{attribute addProperty BoxType "EPP1342-0001-0017"}
{attribute addProperty Id "A_0025_EPP1518_0002_0016EPP1518_7C3C20DE36846A_0026_EPP1518_0002_0017EPP1518_7C3C20DE36846A_0027_EPP1809_0021_0016EPP1809_8059E62316020A_0028_EPP1809_0022_0016EPP1809_8059E62316020A_0029_EPP1819_0021_0016EPP1819_8059E62316020A_0030_EPP1819_0022_0016EPP1819_8059E62316020A_0031_EPP1816_0003_0016EPP1816_9D1B0E2325632A_0032_EPP1816_0008_0016EPP1816_8EE49DA824030A_0033_EPP1816_0008_0017EPP1816_8EE49DA824030A_0034_EPP1816_0008_0018EPP1816_9D1B0E2325632A_0035_EPP1816_3008_0016EPP1816_5F09590E44856"}
{attribute addProperty CRC "1107668744"}
{attribute addProperty SizeInBites "2816"}
{attribute addProperty SizeInBytes "352"}
TYPE A_0024_EPP1342_0001_0017_4205AF08 EXTENDS EPP1342_179A0949 :
STRUCT
	{attribute addProperty Name "A_0025_EPP1518_0002_0016"}
	A_0025_EPP1518_0002_0016 : EPP1518_7C3C20DE;
	{attribute addProperty Name "A_0026_EPP1518_0002_0017"}
	A_0026_EPP1518_0002_0017 : EPP1518_7C3C20DE;
	{attribute addProperty Name "A_0027_EPP1809_0021_0016"}
	A_0027_EPP1809_0021_0016 : EPP1809_8059E623;
	{attribute addProperty Name "A_0028_EPP1809_0022_0016"}
	A_0028_EPP1809_0022_0016 : EPP1809_8059E623;
	{attribute addProperty Name "A_0029_EPP1819_0021_0016"}
	A_0029_EPP1819_0021_0016 : EPP1819_8059E623;
	{attribute addProperty Name "A_0030_EPP1819_0022_0016"}
	A_0030_EPP1819_0022_0016 : EPP1819_8059E623;
	{attribute addProperty Name "A_0031_EPP1816_0003_0016"}
	A_0031_EPP1816_0003_0016 : EPP1816_9D1B0E23;
	{attribute addProperty Name "A_0032_EPP1816_0008_0016"}
	A_0032_EPP1816_0008_0016 : EPP1816_8EE49DA8;
	{attribute addProperty Name "A_0033_EPP1816_0008_0017"}
	A_0033_EPP1816_0008_0017 : EPP1816_8EE49DA8;
	{attribute addProperty Name "A_0034_EPP1816_0008_0018"}
	A_0034_EPP1816_0008_0018 : EPP1816_9D1B0E23;
	{attribute addProperty Name "A_0035_EPP1816_3008_0016"}
	A_0035_EPP1816_3008_0016 : EPP1816_5F09590E;
END_STRUCT
END_TYPE

(* stored: Version 1.2.0.0, ProductVersion 3.1.4024.9
   DUT A_0024_EPP1342_0001_0017_4205AF08: Id {3cad24f5-1bb4-4b6b-bcbd-c2a0e41b7e0f} *)
